// TIA Portal V17 export
// export: Created 2025-03-07T09:24:36.2546827Z, ExportSetting WithDefaults, DisplayName Totally Integrated Automation Portal, DisplayVersion V17 Update 8, DisplayName TIA Portal Openness, DisplayVersion V17 Update 8, DisplayName TIA Portal Version Control Interface, DisplayVersion V17, DisplayName SINAMICS Startdrive Advanced, DisplayVersion V17 SP2, DisplayName SINAMICS Startdrive G110M, G120, G120C, G120D, G120P, G115D, DisplayVersion V17 SP2, DisplayName SINAMICS Startdrive G130, G150, S120, S150, SINAMICS MV, S210, DisplayVersion V17 SP2, DisplayName STEP 7 Professional, DisplayVersion V17 Update 8, DisplayName SINUMERIK ONE STEP 7 Toolbox, DisplayVersion V17 Update 12, DisplayName SINUMERIK 840D sl STEP 7 Toolbox, DisplayVersion V17 Update 12, DisplayName STEP 7 Safety, DisplayVersion V17 Update 6, DisplayName WinCC Advanced, DisplayVersion V17 Update 8
TYPE "FEED HOPPER"
// stored: IsFailsafeCompliant false
   STRUCT
      FAULTED : Bool;   // Faulted
      "START GENERAL CONDITIONS" : Bool;   // Start General Conditions
      "START GENERAL CONDITIONS HELP" : Bool;   // Start General Conditions Help
      "START INITIAL CONDITIONS" : Bool;   // Start Initial Conditions
      "START INITIAL CONDITIONS HELP" : Bool;   // Start Initial Conditions Help
      "START MANUAL REQUEST" : Bool;   // Start Manual Request
      "FEEDBACK ON" : Bool;   // Feedback On
      "START AUTO REQUEST" : Bool;   // Start Auto Request
      "START GLOBAL REQUEST" : Bool;   // Start Global Request
      "START COMMAND" : Bool;   // Start Command
      "SYSTEM ON" : Bool;   // System On
      "STOP GENERAL CONDITIONS" : Bool;   // Stop General Conditions
      "STOP GENERAL CONDITIONS HELP" : Bool;   // Stop General Conditions Help
      "STOP INITIAL CONDITIONS" : Bool;   // Stop Initial Conditions
      "STOP INITIAL CONDITIONS HELP" : Bool;   // Stop Initial Conditions Help
      "STOP MANUAL REQUEST" : Bool;   // Stop Manual Request
      "STOP AUTO REQUEST" : Bool;   // Stop Auto Request
      "STOP GLOBAL REQUEST" : Bool;   // Stop Global Request
      "STOP COMMAND" : Bool;   // Stop Command
      STOPPED : Bool;   // Stopped
      "FEEDBACK OFF" : Bool;   // Feedback Off
   END_STRUCT;
END_TYPE
